// TIA Portal V17 export
// export: Created 2024-08-29T18:23:41.7723351Z, ExportSetting WithDefaults, DisplayName Totally Integrated Automation Portal, DisplayVersion V17 Update 7, DisplayName TIA Portal Openness, DisplayVersion V17 Update 7, DisplayName TIA Portal Version Control Interface, DisplayVersion V17, DisplayName SINAMICS Startdrive Advanced, DisplayVersion V17 SP2, DisplayName SINAMICS Startdrive G110M, G120, G120C, G120D, G120P, G115D, DisplayVersion V17 SP2, DisplayName SINAMICS Startdrive G130, G150, S120, S150, SINAMICS MV, S210, DisplayVersion V17 SP2, DisplayName STEP 7 Professional, DisplayVersion V17 Update 7, DisplayName STEP 7 Safety, DisplayVersion V17 Update 6, DisplayName WinCC Advanced / Unified PC, DisplayVersion V17 Update 7
ORGANIZATION_BLOCK "main"   // OB1, LAD, ProgramCycle
TITLE = "Main Program Sweep (Cycle)"
{ S7_Optimized_Access := 'TRUE' }
VERSION : 0.1
// stored: AutoNumber true, IsIECCheckEnabled false, SetENOAutomatically false
   VAR_INPUT
      Initial_Call : Bool;   // Initial call of this OB
      Remanence : Bool;   // =True, if remanent data are available
   END_VAR
   VAR_TEMP
      BUFFER : String;
   END_VAR
   VAR_TEMP   // added for the SCL form of the ladder/FBD networks
      _w1 : Bool;
      _w2 : Bool;
      _w3 : Bool;
      _w4 : Bool;
      _w5 : Bool;
      _w6 : Bool;
      _w7 : Bool;
      _w8 : Bool;
      _w9 : Bool;
      _w10 : Bool;
   END_VAR
BEGIN

REGION Network 1: SECUENCIA PARA ALARMAR LA MÁQUINA SI SE APAGA A LA MITAD DE UN CICLO DE PRODUCCIÓN
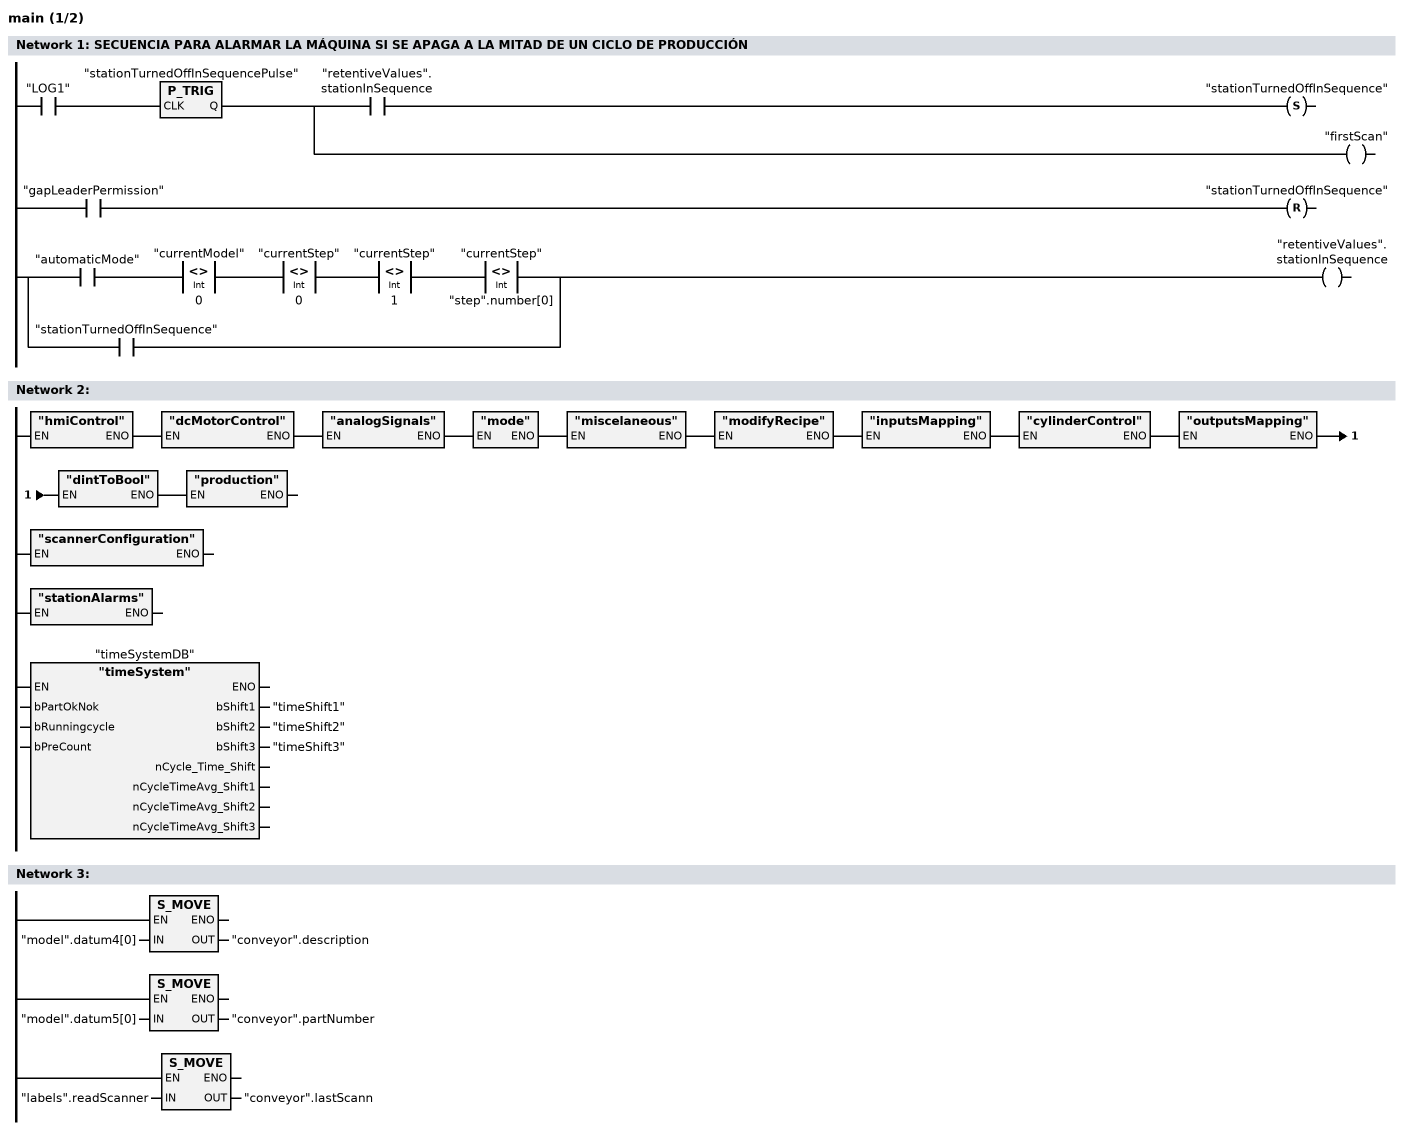
   RUNG wire#powerrail
      Contact( "LOG1" )
      P_Trig( "stationTurnedOffInSequencePulse" )
      wire#w1
      Contact( "retentiveValues".stationInSequence )
      S_Coil( "stationTurnedOffInSequence" )
   END_RUNG
   RUNG wire#w1
      Coil( "firstScan" )
   END_RUNG
   RUNG wire#powerrail
      Contact( "gapLeaderPermission" )
      R_Coil( "stationTurnedOffInSequence" )
   END_RUNG
   RUNG wire#powerrail
      Contact( "automaticMode" )
      { S7_Templates := "SrcType := Int" } NE_Contact(in1 := "currentModel", in2 := 0)
      { S7_Templates := "SrcType := Int" } NE_Contact(in1 := "currentStep", in2 := 0)
      { S7_Templates := "SrcType := Int" } NE_Contact(in1 := "currentStep", in2 := 1)
      { S7_Templates := "SrcType := Int" } NE_Contact(in1 := "currentStep", in2 := "step".number[0])
      wire#w2
      Coil( "retentiveValues".stationInSequence )
   END_RUNG
   RUNG wire#powerrail
      Contact( "stationTurnedOffInSequence" )
   END_RUNG wire#w2
   // the same network as SCL:
   #_w1 := "LOG1" AND NOT "stationTurnedOffInSequencePulse";   // rising edge
   "stationTurnedOffInSequencePulse" := "LOG1";
   IF #_w1 AND "retentiveValues".stationInSequence THEN "stationTurnedOffInSequence" := TRUE; END_IF;
   "firstScan" := #_w1;
   IF "gapLeaderPermission" THEN "stationTurnedOffInSequence" := FALSE; END_IF;
   "retentiveValues".stationInSequence := ("automaticMode" AND ("currentModel" <> 0) AND ("currentStep" <> 0) AND ("currentStep" <> 1) AND ("currentStep" <> "step".number[0])) OR "stationTurnedOffInSequence";
END_REGION

REGION Network 2
   RUNG wire#powerrail
      "hmiControl"()
      "dcMotorControl"()
      "analogSignals"()
      "mode"()
      "miscelaneous"()
      "modifyRecipe"()
      "inputsMapping"()
      "cylinderControl"()
      "outputsMapping"()
      "dintToBool"()
      "production"()
   END_RUNG
   RUNG wire#powerrail
      "scannerConfiguration"()
   END_RUNG
   RUNG wire#powerrail
      "stationAlarms"()
   END_RUNG
   RUNG wire#powerrail
      "timeSystemDB"(bPartOkNok :=, bRunningcycle :=, bPreCount :=, bShift1 => "timeShift1", bShift2 => "timeShift2", bShift3 => "timeShift3", nCycle_Time_Shift =>, nCycleTimeAvg_Shift1 =>, nCycleTimeAvg_Shift2 =>, nCycleTimeAvg_Shift3 =>)
   END_RUNG
   // the same network as SCL:
   "hmiControl"(ENO => #_w1);
   "dcMotorControl"(EN := #_w1, ENO => #_w2);
   "analogSignals"(EN := #_w2, ENO => #_w3);
   "mode"(EN := #_w3, ENO => #_w4);
   "miscelaneous"(EN := #_w4, ENO => #_w5);
   "modifyRecipe"(EN := #_w5, ENO => #_w6);
   "inputsMapping"(EN := #_w6, ENO => #_w7);
   "cylinderControl"(EN := #_w7, ENO => #_w8);
   "outputsMapping"(EN := #_w8, ENO => #_w9);
   "dintToBool"(EN := #_w9, ENO => #_w10);
   IF #_w10 THEN "production"(); END_IF;
   "scannerConfiguration"();
   "stationAlarms"();
   "timeSystemDB"(bShift1 => "timeShift1", bShift2 => "timeShift2", bShift3 => "timeShift3");   // "timeSystem"
END_REGION

REGION Network 3
   RUNG wire#powerrail
      S_Move(in := "model".datum4[0], out => "conveyor".description)
   END_RUNG
   RUNG wire#powerrail
      S_Move(in := "model".datum5[0], out => "conveyor".partNumber)
   END_RUNG
   RUNG wire#powerrail
      S_Move(in := "labels".readScanner, out => "conveyor".lastScann)
   END_RUNG
   // the same network as SCL:
   "conveyor".description := "model".datum4[0];
   "conveyor".partNumber := "model".datum5[0];
   "conveyor".lastScann := "labels".readScanner;
END_REGION

REGION Network 4: Permissions
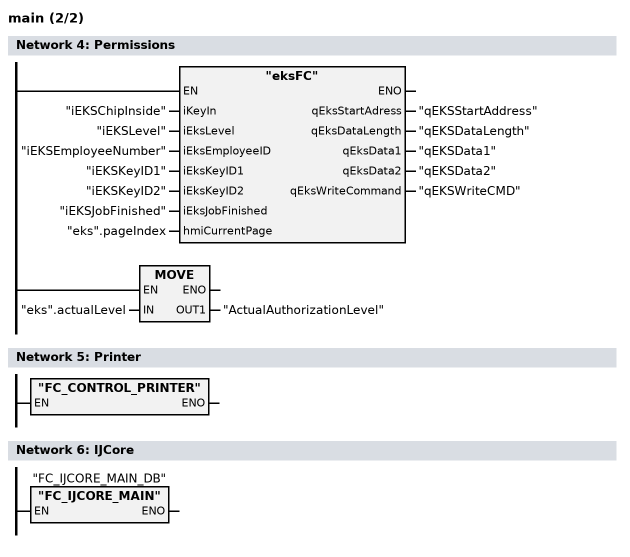
   RUNG wire#powerrail
      "eksFC"(iKeyIn := "iEKSChipInside", iEksLevel := "iEKSLevel", iEksEmployeeID := "iEKSEmployeeNumber", iEksKeyID1 := "iEKSKeyID1", iEksKeyID2 := "iEKSKeyID2", iEksJobFinished := "iEKSJobFinished", hmiCurrentPage := "eks".pageIndex, qEksStartAdress => "qEKSStartAddress", qEksDataLength => "qEKSDataLength", qEksData1 => "qEKSData1", qEksData2 => "qEKSData2", qEksWriteCommand => "qEKSWriteCMD")
   END_RUNG
   RUNG wire#powerrail
      Move(in := "eks".actualLevel, out1 => "ActualAuthorizationLevel")
   END_RUNG
   // the same network as SCL:
   "eksFC"(iKeyIn := "iEKSChipInside",
           iEksLevel := "iEKSLevel",
           iEksEmployeeID := "iEKSEmployeeNumber",
           iEksKeyID1 := "iEKSKeyID1",
           iEksKeyID2 := "iEKSKeyID2",
           iEksJobFinished := "iEKSJobFinished",
           hmiCurrentPage := "eks".pageIndex,
           qEksStartAdress => "qEKSStartAddress",
           qEksDataLength => "qEKSDataLength",
           qEksData1 => "qEKSData1",
           qEksData2 => "qEKSData2",
           qEksWriteCommand => "qEKSWriteCMD");
   "ActualAuthorizationLevel" := "eks".actualLevel;
END_REGION

REGION Network 5: Printer
   RUNG wire#powerrail
      "FC_CONTROL_PRINTER"()
   END_RUNG
   // the same network as SCL:
   "FC_CONTROL_PRINTER"();
END_REGION

REGION Network 6: IJCore
   RUNG wire#powerrail
      "FC_IJCORE_MAIN_DB"()
   END_RUNG
   // the same network as SCL:
   "FC_IJCORE_MAIN_DB"();   // "FC_IJCORE_MAIN"
END_REGION
END_ORGANIZATION_BLOCK
